Yaskawa INFORM job: u_profile_cylinder_program.JBI

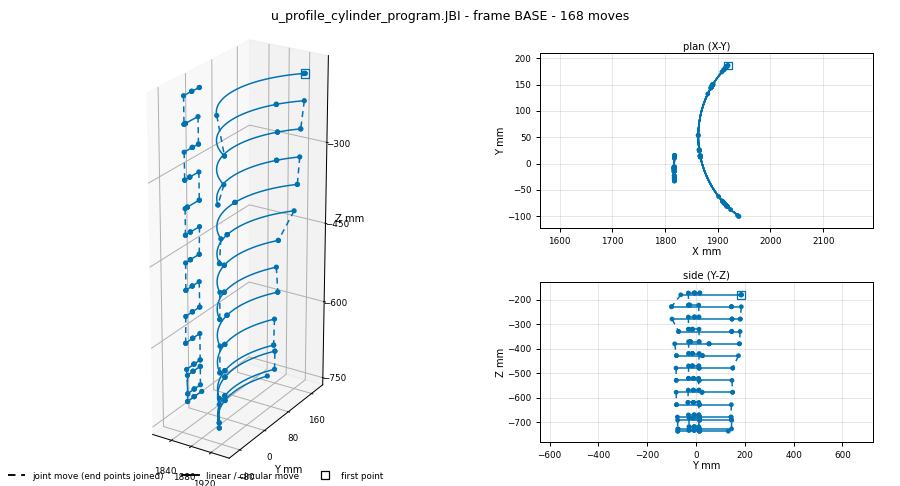
[picture p0: tool path of u_profile_cylinder_program.JBI in frame BASE, 168 of 229 moves have a stored position in this frame; points joined in program order, loops and branches not executed]
/JOB
//NAME u_profile_cylinder_program
//POS
///NPOS 224,0,224,0,0,0
///TOOL 0
///POSTYPE BASE
///RECTAN
///RCONF 0,0,0,0,0,0,0,0,0,0,0,0,0,0,0,0,0,0,0,0,0,0,0,0
C00000=1919.318375,186.161452,-178.861000,134.506550,-89.999999,5.000000
C00001=1919.318375,186.161452,-178.861000,134.506550,-89.999999,5.000000
C00002=1918.589363,185.440980,-178.861000,134.818396,-90.000000,5.000000
C00003=1917.365275,184.213378,-178.861000,135.345852,-89.999999,5.000000
C00004=1917.365275,184.213378,-178.861000,135.345852,-89.999999,5.000000
C00005=1917.365275,184.213378,-178.861000,135.345852,-89.999999,5.000000
C00006=1888.696320,146.804587,-178.861000,149.723241,-90.000000,5.000000
C00007=1901.530648,-62.264651,-178.861000,-142.697519,-90.000000,5.000000
C00008=1940.003397,-100.029578,-227.659000,-126.238595,-90.000000,5.000000
C00009=1940.003397,-100.029578,-227.659000,-126.238595,-90.000000,5.000000
C00010=1900.428189,-60.802911,-227.659000,-143.254569,-90.000000,5.000000
C00011=1887.843950,145.329282,-227.659000,150.241639,-90.000000,5.000000
C00012=1887.843950,145.329282,-227.659000,150.241639,-90.000000,5.000000
C00013=1887.843950,145.329282,-227.659000,150.241639,-90.000000,5.000000
C00014=1916.985731,183.828118,-227.659000,135.510396,-90.000000,5.000000
C00015=1918.736080,185.586610,-227.659000,134.755500,-90.000000,5.000000
C00016=1914.779750,181.544281,-278.103500,136.476486,-90.000000,5.000000
C00017=1914.779750,181.544281,-278.103500,136.476486,-90.000000,5.000000
C00018=1892.910079,153.679854,-278.103500,147.269621,-90.000000,5.000000
C00019=1889.143474,147.566403,-278.103500,149.454479,-90.000000,5.000000
C00020=1889.143474,147.566403,-278.103500,149.454479,-90.000000,5.000000
C00021=1889.143474,147.566403,-278.103500,149.454479,-90.000000,5.000000
C00022=1888.389247,146.276640,-278.103500,149.909065,-89.999999,5.000000
C00023=1937.546390,-98.197860,-278.103500,-127.171032,-89.999999,5.000000
C00024=1908.746745,-71.161367,-329.209500,-139.211685,-90.000000,5.000000
C00025=1908.746745,-71.161367,-329.209500,-139.211685,-90.000000,5.000000
C00026=1863.944997,70.602477,-329.209500,174.287971,-90.000000,5.000000
C00027=1888.494246,146.457607,-329.209500,149.845409,-90.000000,5.000000
C00028=1888.494246,146.457607,-329.209500,149.845409,-90.000000,5.000000
C00029=1888.494246,146.457607,-329.209500,149.845409,-90.000000,5.000000
C00030=1912.550325,179.155729,-329.209500,137.470595,-90.000000,5.000000
C00031=1913.986749,180.704173,-329.209500,136.827978,-90.000000,5.000000
C00032=1911.467631,177.965220,-379.550000,137.960200,-89.999999,5.000000
C00033=1911.467631,177.965220,-379.550000,137.960200,-89.999999,5.000000
C00034=1880.825526,131.812975,-379.550000,154.876624,-90.000000,5.000000
C00035=1863.018641,53.669024,-379.550000,175.000000,-90.000000,5.000000
C00036=1863.018641,53.669024,-379.550000,175.000000,-90.000000,5.000000
C00037=1863.018641,53.669024,-379.550000,175.000000,-90.000000,5.000000
C00038=1873.111078,-8.987699,-379.550000,-161.148807,-90.000000,5.000000
C00039=1924.416941,-87.270246,-379.550000,-132.370057,-90.000000,5.000000
C00040=1916.910765,-80.032620,-428.210500,-135.542952,-89.999999,5.000000
C00041=1916.910765,-80.032620,-428.210500,-135.542952,-89.999999,5.000000
C00042=1880.533893,-27.468951,-428.210500,-155.086432,-90.000000,5.000000
C00043=1864.757197,26.266217,-428.210500,-172.188992,-90.000000,5.000000
C00044=1864.757197,26.266217,-428.210500,-172.188992,-90.000000,5.000000
C00045=1864.757197,26.266217,-428.210500,-172.188992,-90.000000,5.000000
C00046=1866.619713,88.554638,-428.210500,168.763556,-90.000000,5.000000
C00047=1907.955855,173.957872,-428.210500,139.581419,-90.000000,5.000000
C00048=1890.844588,150.392245,-479.170000,148.450933,-90.000000,5.000000
C00049=1890.844588,150.392245,-479.170000,148.450933,-90.000000,5.000000
C00050=1866.110873,85.893326,-479.170000,169.587940,-90.000000,5.000000
C00051=1867.114547,12.756098,-479.170000,-168.015481,-90.000000,5.000000
C00052=1867.114547,12.756098,-479.170000,-168.015481,-90.000000,5.000000
C00053=1867.114547,12.756098,-479.170000,-168.015481,-90.000000,5.000000
C00054=1885.121266,-36.678278,-479.170000,-151.955707,-89.999999,5.000000
C00055=1918.627673,-81.759895,-479.170000,-134.801966,-90.000000,5.000000
C00056=1917.564533,-80.695611,-529.349500,-135.259659,-90.000000,5.000000
C00057=1917.564533,-80.695611,-529.349500,-135.259659,-90.000000,5.000000
C00058=1884.758137,-35.993208,-529.349500,-152.191612,-89.999999,5.000000
C00059=1867.109072,12.781899,-529.349500,-168.023506,-89.999999,5.000000
C00060=1867.109072,12.781899,-529.349500,-168.023506,-89.999999,5.000000
C00061=1867.109072,12.781899,-529.349500,-168.023506,-89.999999,5.000000
C00062=1865.977888,85.161474,-529.349500,169.814254,-90.000000,5.000000
C00063=1889.033377,147.379588,-529.349500,149.520454,-90.000000,5.000000
C00064=1890.657657,150.087139,-578.090000,148.559800,-89.999999,5.000000
C00065=1890.657657,150.087139,-578.090000,148.559800,-89.999999,5.000000
C00066=1866.130659,86.000828,-578.090000,169.554683,-90.000000,5.000000
C00067=1865.001154,24.546756,-578.090000,-171.660601,-90.000000,5.000000
C00068=1865.001154,24.546756,-578.090000,-171.660601,-90.000000,5.000000
C00069=1865.001154,24.546756,-578.090000,-171.660601,-90.000000,5.000000
C00070=1880.545792,-27.494565,-578.090000,-155.077839,-89.999999,5.000000
C00071=1918.072525,-81.206271,-578.090000,-135.040507,-90.000000,5.000000
C00072=1916.577251,-79.691863,-629.004000,-135.688022,-90.000000,5.000000
C00073=1916.577251,-79.691863,-629.004000,-135.688022,-90.000000,5.000000
C00074=1884.660871,-35.808545,-629.004000,-152.255114,-90.000000,5.000000
C00075=1866.788899,14.322936,-629.004000,-168.502384,-90.000000,5.000000
C00076=1866.788899,14.322936,-629.004000,-168.502384,-90.000000,5.000000
C00077=1866.788899,14.322936,-629.004000,-168.502384,-90.000000,5.000000
C00078=1866.111622,85.897399,-629.004000,169.586680,-90.000000,5.000000
C00079=1887.536562,144.789584,-629.004000,150.430609,-90.000000,5.000000
C00080=1886.887686,143.636513,-679.693000,150.833168,-89.999999,5.000000
C00081=1886.887686,143.636513,-679.693000,150.833168,-89.999999,5.000000
C00082=1865.941224,84.956765,-679.693000,169.877528,-89.999999,5.000000
C00083=1866.729376,14.616759,-679.693000,-168.593596,-90.000000,5.000000
C00084=1866.729376,14.616759,-679.693000,-168.593596,-90.000000,5.000000
C00085=1866.729376,14.616759,-679.693000,-168.593596,-90.000000,5.000000
C00086=1884.804416,-36.080897,-679.693000,-152.161445,-89.999999,5.000000
C00087=1913.224618,-76.167805,-679.693000,-137.167966,-90.000000,5.000000
C00088=1911.184789,-73.931681,-728.214500,-138.088869,-90.000000,5.000000
C00089=1911.184789,-73.931681,-728.214500,-138.088869,-90.000000,5.000000
C00090=1884.746150,-35.970477,-728.214500,-152.199431,-89.999999,5.000000
C00091=1866.919433,13.686824,-728.214500,-168.304812,-90.000000,5.000000
C00092=1866.919433,13.686824,-728.214500,-168.304812,-90.000000,5.000000
C00093=1866.919433,13.686824,-728.214500,-168.304812,-90.000000,5.000000
C00094=1865.765968,83.959631,-728.214500,170.185559,-89.999999,5.000000
C00095=1887.960264,145.532429,-728.214500,150.170417,-90.000000,5.000000
C00096=1888.186604,145.926067,-692.282460,175.000000,-60.000000,-29.967735
C00097=1888.186604,145.926067,-692.282460,175.000000,-60.000000,-29.967735
C00098=1865.952407,85.019339,-692.282460,175.000000,-60.000000,-10.141812
C00099=1866.711119,14.707370,-692.282460,175.000000,-60.000000,11.378282
C00100=1866.711119,14.707370,-692.282460,175.000000,-60.000000,11.378282
C00101=1866.711119,14.707370,-692.282460,175.000000,-60.000000,11.378282
C00102=1884.830220,-36.129742,-692.282460,-175.000000,-60.000000,27.855362
C00103=1912.302833,-75.166247,-692.282460,-175.000000,-60.000000,42.417891
C00104=1911.869257,-74.690086,-737.636460,175.000000,-60.000000,42.221957
C00105=1911.869257,-74.690086,-737.636460,175.000000,-60.000000,42.221957
C00106=1884.879767,-36.223432,-737.636460,175.000000,-60.000000,27.887609
C00107=1866.818502,14.177698,-737.636460,175.000000,-60.000000,11.542714
C00108=1866.818502,14.177698,-737.636460,175.000000,-60.000000,11.542714
C00109=1866.818502,14.177698,-737.636460,175.000000,-60.000000,11.542714
C00110=1864.683098,76.906826,-737.636460,175.000000,-60.000000,-7.643334
C00111=1881.053412,132.297152,-737.636460,175.000000,-60.000000,-25.286189
C00112=1817.990504,15.588637,-171.217500,175.000000,-89.999999,5.000000
C00113=1817.990504,15.588637,-171.217500,175.000000,-89.999999,5.000000
C00114=1817.535552,3.881759,-171.217500,175.000000,-90.000000,5.000000
C00115=1817.349789,-6.442676,-171.217500,175.000000,-90.000000,5.000000
C00116=1817.349789,-6.442676,-171.217500,175.000000,-90.000000,5.000000
C00117=1817.349789,-6.442676,-171.217500,175.000000,-90.000000,5.000000
C00118=1817.526814,-25.140198,-171.217500,-175.000000,-90.000000,5.000000
C00119=1817.723727,-31.135669,-171.217500,-175.000000,-90.000000,5.000000
C00120=1817.711525,-30.816430,-220.926500,-175.000000,-90.000000,5.000000
C00121=1817.711525,-30.816430,-220.926500,-175.000000,-90.000000,5.000000
C00122=1817.677190,-29.889507,-220.926500,-175.000000,-89.999999,5.000000
C00123=1817.559266,-26.288875,-220.926500,-175.000000,-89.999999,5.000000
C00124=1817.559266,-26.288875,-220.926500,-175.000000,-89.999999,5.000000
C00125=1817.559266,-26.288875,-220.926500,-175.000000,-89.999999,5.000000
C00126=1817.458554,-22.357350,-220.926500,-175.000000,-90.000000,5.000000
C00127=1817.791962,11.259122,-220.926500,175.000000,-89.999999,5.000000
C00128=1817.818806,11.892960,-269.769000,175.000000,-90.000000,5.000000
C00129=1817.818806,11.892960,-269.769000,175.000000,-90.000000,5.000000
C00130=1817.515491,3.140532,-269.769000,175.000000,-90.000000,5.000000
C00131=1817.353005,-6.067748,-269.769000,175.000000,-89.999999,5.000000
C00132=1817.353005,-6.067748,-269.769000,175.000000,-89.999999,5.000000
C00133=1817.353005,-6.067748,-269.769000,175.000000,-89.999999,5.000000
C00134=1817.536459,-25.490982,-269.769000,-175.000000,-89.999999,5.000000
C00135=1817.725812,-31.189730,-269.769000,-175.000000,-89.999999,5.000000
C00136=1817.698334,-30.465502,-319.757000,-175.000000,-89.999999,5.000000
C00137=1817.698334,-30.465502,-319.757000,-175.000000,-89.999999,5.000000
C00138=1817.564494,-26.466058,-319.757000,-175.000000,-89.999999,5.000000
C00139=1817.346049,-14.652350,-319.757000,-175.000000,-90.000000,5.000000
C00140=1817.346049,-14.652350,-319.757000,-175.000000,-90.000000,5.000000
C00141=1817.346049,-14.652350,-319.757000,-175.000000,-90.000000,5.000000
C00142=1817.456468,0.685090,-319.757000,175.000000,-90.000000,5.000000
C00143=1817.843348,12.457295,-319.757000,175.000000,-89.999999,5.000000
C00144=1817.862419,12.886540,-370.985000,175.000000,-89.999999,5.000000
C00145=1817.862419,12.886540,-370.985000,175.000000,-89.999999,5.000000
C00146=1817.718241,9.416200,-370.985000,175.000000,-89.999999,5.000000
C00147=1817.468232,-22.791229,-370.985000,-175.000000,-90.000000,5.000000
C00148=1817.468232,-22.791229,-370.985000,-175.000000,-90.000000,5.000000
C00149=1817.468232,-22.791229,-370.985000,-175.000000,-90.000000,5.000000
C00150=1817.608303,-27.878641,-370.985000,-175.000000,-90.000000,5.000000
C00151=1817.689997,-30.240415,-370.985000,-175.000000,-90.000000,5.000000
C00152=1817.677729,-29.904397,-419.370500,-175.000000,-90.000000,5.000000
C00153=1817.677729,-29.904397,-419.370500,-175.000000,-90.000000,5.000000
C00154=1817.565488,-26.499532,-419.370500,-175.000000,-90.000000,5.000000
C00155=1817.344102,-14.376187,-419.370500,-175.000000,-89.999999,5.000000
C00156=1817.344102,-14.376187,-419.370500,-175.000000,-89.999999,5.000000
C00157=1817.344102,-14.376187,-419.370500,-175.000000,-89.999999,5.000000
C00158=1817.497248,2.430436,-419.370500,175.000000,-89.999999,5.000000
C00159=1817.865089,12.946001,-419.370500,175.000000,-90.000000,5.000000
C00160=1817.804165,11.549491,-470.057500,175.000000,-90.000000,5.000000
C00161=1817.804165,11.549491,-470.057500,175.000000,-90.000000,5.000000
C00162=1817.398164,-2.420661,-470.057500,175.000000,-89.999999,5.000000
C00163=1817.348154,-14.930333,-470.057500,-175.000000,-89.999999,5.000000
C00164=1817.348154,-14.930333,-470.057500,-175.000000,-89.999999,5.000000
C00165=1817.348154,-14.930333,-470.057500,-175.000000,-89.999999,5.000000
C00166=1817.479346,-23.270935,-470.057500,-175.000000,-89.999999,5.000000
C00167=1817.696262,-30.409800,-470.057500,-175.000000,-90.000000,5.000000
C00168=1817.702789,-30.584713,-520.961000,-175.000000,-89.999999,5.000000
C00169=1817.702789,-30.584713,-520.961000,-175.000000,-89.999999,5.000000
C00170=1817.473301,-23.012345,-520.961000,-175.000000,-89.999999,5.000000
C00171=1817.332146,-10.303971,-520.961000,175.000000,-89.999999,5.000000
C00172=1817.332146,-10.303971,-520.961000,175.000000,-89.999999,5.000000
C00173=1817.332146,-10.303971,-520.961000,175.000000,-89.999999,5.000000
C00174=1817.481924,1.803009,-520.961000,175.000000,-90.000000,5.000000
C00175=1817.771654,10.767186,-520.961000,175.000000,-90.000000,5.000000
C00176=1817.807943,11.638625,-569.380500,175.000000,-89.999999,5.000000
C00177=1817.807943,11.638625,-569.380500,175.000000,-89.999999,5.000000
C00178=1817.492353,2.233288,-569.380500,175.000000,-90.000000,5.000000
C00179=1817.332011,-10.484289,-569.380500,175.000000,-89.999999,5.000000
C00180=1817.332011,-10.484289,-569.380500,175.000000,-89.999999,5.000000
C00181=1817.332011,-10.484289,-569.380500,175.000000,-89.999999,5.000000
C00182=1817.402898,-19.449712,-569.380500,-175.000000,-90.000000,5.000000
C00183=1817.753185,-31.886429,-569.380500,-175.000000,-90.000000,5.000000
C00184=1817.797491,-32.967741,-619.760000,-175.000000,-90.000000,5.000000
C00185=1817.797491,-32.967741,-619.760000,-175.000000,-90.000000,5.000000
C00186=1817.408869,-19.806675,-619.760000,-175.000000,-90.000000,5.000000
C00187=1817.332035,-10.445182,-619.760000,175.000000,-90.000000,5.000000
C00188=1817.332035,-10.445182,-619.760000,175.000000,-90.000000,5.000000
C00189=1817.332035,-10.445182,-619.760000,175.000000,-90.000000,5.000000
C00190=1817.487025,2.015284,-619.760000,175.000000,-90.000000,5.000000
C00191=1817.799497,11.438868,-619.760000,175.000000,-90.000000,5.000000
C00192=1817.816514,11.839522,-670.886500,175.000000,-90.000000,5.000000
C00193=1817.816514,11.839522,-670.886500,175.000000,-90.000000,5.000000
C00194=1817.497087,2.424002,-670.886500,175.000000,-89.999999,5.000000
C00195=1817.343542,-7.283868,-670.886500,175.000000,-90.000000,5.000000
C00196=1817.343542,-7.283868,-670.886500,175.000000,-90.000000,5.000000
C00197=1817.343542,-7.283868,-670.886500,175.000000,-90.000000,5.000000
C00198=1817.403330,-19.476025,-670.886500,-175.000000,-89.999999,5.000000
C00199=1817.714379,-30.891550,-670.886500,-175.000000,-90.000000,5.000000
C00200=1817.617890,-28.172449,-719.382000,-175.000000,-89.999999,5.000000
C00201=1817.617890,-28.172449,-719.382000,-175.000000,-89.999999,5.000000
C00202=1817.404390,-19.540283,-719.382000,-175.000000,-90.000000,5.000000
C00203=1817.344900,-7.084679,-719.382000,175.000000,-89.999999,5.000000
C00204=1817.344900,-7.084679,-719.382000,175.000000,-89.999999,5.000000
C00205=1817.344900,-7.084679,-719.382000,175.000000,-89.999999,5.000000
C00206=1817.490538,2.159410,-719.382000,175.000000,-89.999999,5.000000
C00207=1817.819284,11.904095,-719.382000,175.000000,-89.999999,5.000000
C00208=1817.821861,11.963975,-683.466460,175.000000,-60.000000,-5.000000
C00209=1817.821861,11.963975,-683.466460,175.000000,-60.000000,-5.000000
C00210=1817.474996,1.508823,-683.466460,-175.000000,-60.000000,-5.000000
C00211=1817.332124,-10.329006,-683.466460,175.000000,-60.000000,-5.000000
C00212=1817.332124,-10.329006,-683.466460,175.000000,-60.000000,-5.000000
C00213=1817.332124,-10.329006,-683.466460,175.000000,-60.000000,-5.000000
C00214=1817.403522,-19.487738,-683.466460,175.000000,-60.000000,5.000000
C00215=1817.622059,-28.298669,-683.466460,175.000000,-60.000000,5.000000
C00216=1817.637760,-28.766095,-734.096960,175.000000,-60.000000,5.000000
C00217=1817.637760,-28.766095,-734.096960,175.000000,-60.000000,5.000000
C00218=1817.405775,-19.623546,-734.096960,-175.000000,-60.000000,5.000000
C00219=1817.341568,-7.595472,-734.096960,-175.000000,-60.000000,-5.000000
C00220=1817.341568,-7.595472,-734.096960,-175.000000,-60.000000,-5.000000
C00221=1817.341568,-7.595472,-734.096960,-175.000000,-60.000000,-5.000000
C00222=1817.484869,1.925964,-734.096960,-175.000000,-60.000000,-5.000000
C00223=1817.997034,15.719000,-734.096960,175.000000,-60.000000,-5.000000
///POSTYPE PULSE
///PULSE
EX00000=261120.0
EX00001=362496.0
///POSTYPE PULSE
///PULSE
EC00000=261120.0
EC00001=261120.0
EC00002=261120.0
EC00003=261120.0
EC00004=261120.0
EC00005=261120.0
EC00006=261120.0
EC00007=261120.0
EC00008=261120.0
EC00009=261120.0
EC00010=261120.0
EC00011=261120.0
EC00012=261120.0
EC00013=261120.0
EC00014=261120.0
EC00015=261120.0
EC00016=261120.0
EC00017=261120.0
EC00018=261120.0
EC00019=261120.0
EC00020=261120.0
EC00021=261120.0
EC00022=261120.0
EC00023=261120.0
EC00024=261120.0
EC00025=261120.0
EC00026=261120.0
EC00027=261120.0
EC00028=261120.0
EC00029=261120.0
EC00030=261120.0
EC00031=261120.0
EC00032=261120.0
EC00033=261120.0
EC00034=261120.0
EC00035=261120.0
EC00036=261120.0
EC00037=261120.0
EC00038=261120.0
EC00039=261120.0
EC00040=261120.0
EC00041=261120.0
EC00042=261120.0
EC00043=261120.0
EC00044=261120.0
EC00045=261120.0
EC00046=261120.0
EC00047=261120.0
EC00048=261120.0
EC00049=261120.0
EC00050=261120.0
EC00051=261120.0
EC00052=261120.0
EC00053=261120.0
EC00054=261120.0
EC00055=261120.0
EC00056=261120.0
EC00057=261120.0
EC00058=261120.0
EC00059=261120.0
EC00060=261120.0
EC00061=261120.0
EC00062=261120.0
EC00063=261120.0
EC00064=261120.0
EC00065=261120.0
EC00066=261120.0
EC00067=261120.0
EC00068=261120.0
EC00069=261120.0
EC00070=261120.0
EC00071=261120.0
EC00072=261120.0
EC00073=261120.0
EC00074=261120.0
EC00075=261120.0
EC00076=261120.0
EC00077=261120.0
EC00078=261120.0
EC00079=261120.0
EC00080=261120.0
EC00081=261120.0
EC00082=261120.0
EC00083=261120.0
EC00084=261120.0
EC00085=261120.0
EC00086=261120.0
EC00087=261120.0
EC00088=261120.0
EC00089=261120.0
EC00090=261120.0
EC00091=261120.0
EC00092=261120.0
EC00093=261120.0
EC00094=261120.0
EC00095=261120.0
EC00096=261120.0
EC00097=261120.0
EC00098=261120.0
EC00099=261120.0
EC00100=261120.0
EC00101=261120.0
EC00102=261120.0
EC00103=261120.0
EC00104=261120.0
EC00105=261120.0
EC00106=261120.0
EC00107=261120.0
EC00108=261120.0
EC00109=261120.0
EC00110=261120.0
EC00111=261120.0
EC00112=362496.0
EC00113=362496.0
EC00114=362496.0
EC00115=362496.0
EC00116=362496.0
EC00117=362496.0
EC00118=362496.0
EC00119=362496.0
EC00120=362496.0
EC00121=362496.0
EC00122=362496.0
EC00123=362496.0
EC00124=362496.0
EC00125=362496.0
EC00126=362496.0
EC00127=362496.0
EC00128=362496.0
EC00129=362496.0
EC00130=362496.0
EC00131=362496.0
EC00132=362496.0
EC00133=362496.0
EC00134=362496.0
EC00135=362496.0
EC00136=362496.0
EC00137=362496.0
EC00138=362496.0
EC00139=362496.0
EC00140=362496.0
EC00141=362496.0
EC00142=362496.0
EC00143=362496.0
EC00144=362496.0
EC00145=362496.0
EC00146=362496.0
EC00147=362496.0
EC00148=362496.0
EC00149=362496.0
EC00150=362496.0
EC00151=362496.0
EC00152=362496.0
EC00153=362496.0
EC00154=362496.0
EC00155=362496.0
EC00156=362496.0
EC00157=362496.0
EC00158=362496.0
EC00159=362496.0
EC00160=362496.0
EC00161=362496.0
EC00162=362496.0
EC00163=362496.0
EC00164=362496.0
EC00165=362496.0
EC00166=362496.0
EC00167=362496.0
EC00168=362496.0
EC00169=362496.0
EC00170=362496.0
EC00171=362496.0
EC00172=362496.0
EC00173=362496.0
EC00174=362496.0
EC00175=362496.0
EC00176=362496.0
EC00177=362496.0
EC00178=362496.0
EC00179=362496.0
EC00180=362496.0
EC00181=362496.0
EC00182=362496.0
EC00183=362496.0
EC00184=362496.0
EC00185=362496.0
EC00186=362496.0
EC00187=362496.0
EC00188=362496.0
EC00189=362496.0
EC00190=362496.0
EC00191=362496.0
EC00192=362496.0
EC00193=362496.0
EC00194=362496.0
EC00195=362496.0
EC00196=362496.0
EC00197=362496.0
EC00198=362496.0
EC00199=362496.0
EC00200=362496.0
EC00201=362496.0
EC00202=362496.0
EC00203=362496.0
EC00204=362496.0
EC00205=362496.0
EC00206=362496.0
EC00207=362496.0
EC00208=362496.0
EC00209=362496.0
EC00210=362496.0
EC00211=362496.0
EC00212=362496.0
EC00213=362496.0
EC00214=362496.0
EC00215=362496.0
EC00216=362496.0
EC00217=362496.0
EC00218=362496.0
EC00219=362496.0
EC00220=362496.0
EC00221=362496.0
EC00222=362496.0
EC00223=362496.0
//INST
///DATE 2023/08/16 15:26
///ATTR SC,RW,RJ
////FRAME BASE
///GROUP1 RB1,ST1
NOP
MOVJ P009 EX000 VJ=15.00
MOVJ C00000 EC00000 VJ=15.0
CALL JOB:SPYON
MOVC C00001 EC00001 V=150.0
MOVC C00002 EC00002 V=150.0
MOVC C00003 EC00003 V=150.0
MOVJ C00004 EC00004 VJ=15.0
MOVC C00005 EC00005 V=150.0
MOVC C00006 EC00006 V=150.0
MOVC C00007 EC00007 V=150.0
MOVJ C00008 EC00008 VJ=15.0
MOVC C00009 EC00009 V=150.0
MOVC C00010 EC00010 V=150.0
MOVC C00011 EC00011 V=150.0
MOVJ C00012 EC00012 VJ=15.0
MOVC C00013 EC00013 V=150.0
MOVC C00014 EC00014 V=150.0
MOVC C00015 EC00015 V=150.0
MOVJ C00016 EC00016 VJ=15.0
MOVC C00017 EC00017 V=150.0
MOVC C00018 EC00018 V=150.0
MOVC C00019 EC00019 V=150.0
MOVJ C00020 EC00020 VJ=15.0
MOVC C00021 EC00021 V=150.0
MOVC C00022 EC00022 V=150.0
MOVC C00023 EC00023 V=150.0
MOVJ C00024 EC00024 VJ=15.0
MOVC C00025 EC00025 V=150.0
MOVC C00026 EC00026 V=150.0
MOVC C00027 EC00027 V=150.0
MOVJ C00028 EC00028 VJ=15.0
MOVC C00029 EC00029 V=150.0
MOVC C00030 EC00030 V=150.0
MOVC C00031 EC00031 V=150.0
MOVJ C00032 EC00032 VJ=15.0
MOVC C00033 EC00033 V=150.0
MOVC C00034 EC00034 V=150.0
MOVC C00035 EC00035 V=150.0
MOVJ C00036 EC00036 VJ=15.0
MOVC C00037 EC00037 V=150.0
MOVC C00038 EC00038 V=150.0
MOVC C00039 EC00039 V=150.0
MOVJ C00040 EC00040 VJ=15.0
MOVC C00041 EC00041 V=150.0
MOVC C00042 EC00042 V=150.0
MOVC C00043 EC00043 V=150.0
MOVJ C00044 EC00044 VJ=15.0
MOVC C00045 EC00045 V=150.0
MOVC C00046 EC00046 V=150.0
MOVC C00047 EC00047 V=150.0
MOVJ C00048 EC00048 VJ=15.0
MOVC C00049 EC00049 V=150.0
MOVC C00050 EC00050 V=150.0
MOVC C00051 EC00051 V=150.0
MOVJ C00052 EC00052 VJ=15.0
MOVC C00053 EC00053 V=150.0
MOVC C00054 EC00054 V=150.0
MOVC C00055 EC00055 V=150.0
MOVJ C00056 EC00056 VJ=15.0
MOVC C00057 EC00057 V=150.0
MOVC C00058 EC00058 V=150.0
MOVC C00059 EC00059 V=150.0
MOVJ C00060 EC00060 VJ=15.0
MOVC C00061 EC00061 V=150.0
MOVC C00062 EC00062 V=150.0
MOVC C00063 EC00063 V=150.0
MOVJ C00064 EC00064 VJ=15.0
MOVC C00065 EC00065 V=150.0
MOVC C00066 EC00066 V=150.0
MOVC C00067 EC00067 V=150.0
MOVJ C00068 EC00068 VJ=15.0
MOVC C00069 EC00069 V=150.0
MOVC C00070 EC00070 V=150.0
MOVC C00071 EC00071 V=150.0
MOVJ C00072 EC00072 VJ=15.0
MOVC C00073 EC00073 V=150.0
MOVC C00074 EC00074 V=150.0
MOVC C00075 EC00075 V=150.0
MOVJ C00076 EC00076 VJ=15.0
MOVC C00077 EC00077 V=150.0
MOVC C00078 EC00078 V=150.0
MOVC C00079 EC00079 V=150.0
MOVJ C00080 EC00080 VJ=15.0
MOVC C00081 EC00081 V=150.0
MOVC C00082 EC00082 V=150.0
MOVC C00083 EC00083 V=150.0
MOVJ C00084 EC00084 VJ=15.0
MOVC C00085 EC00085 V=150.0
MOVC C00086 EC00086 V=150.0
MOVC C00087 EC00087 V=150.0
MOVJ C00088 EC00088 VJ=15.0
MOVC C00089 EC00089 V=150.0
MOVC C00090 EC00090 V=150.0
MOVC C00091 EC00091 V=150.0
MOVJ C00092 EC00092 VJ=15.0
MOVC C00093 EC00093 V=150.0
MOVC C00094 EC00094 V=150.0
MOVC C00095 EC00095 V=150.0
MOVJ C00096 EC00096 VJ=15.0
MOVC C00097 EC00097 V=150.0
MOVC C00098 EC00098 V=150.0
MOVC C00099 EC00099 V=150.0
MOVJ C00100 EC00100 VJ=15.0
MOVC C00101 EC00101 V=150.0
MOVC C00102 EC00102 V=150.0
MOVC C00103 EC00103 V=150.0
MOVJ C00104 EC00104 VJ=15.0
MOVC C00105 EC00105 V=150.0
MOVC C00106 EC00106 V=150.0
MOVC C00107 EC00107 V=150.0
MOVJ C00108 EC00108 VJ=15.0
MOVC C00109 EC00109 V=150.0
MOVC C00110 EC00110 V=150.0
MOVC C00111 EC00111 V=150.0
CALL JOB:SPYOF
MOVJ P009 VJ=15.00
MOVL P009 EX00000 V=150.0
MOVJ C00112 EC00112 VJ=15.0
CALL JOB:SPYON
MOVC C00113 EC00113 V=150.0
MOVC C00114 EC00114 V=150.0
MOVC C00115 EC00115 V=150.0
MOVJ C00116 EC00116 VJ=15.0
MOVC C00117 EC00117 V=150.0
MOVC C00118 EC00118 V=150.0
MOVC C00119 EC00119 V=150.0
MOVJ C00120 EC00120 VJ=15.0
MOVC C00121 EC00121 V=150.0
MOVC C00122 EC00122 V=150.0
MOVC C00123 EC00123 V=150.0
MOVJ C00124 EC00124 VJ=15.0
MOVC C00125 EC00125 V=150.0
MOVC C00126 EC00126 V=150.0
MOVC C00127 EC00127 V=150.0
MOVJ C00128 EC00128 VJ=15.0
MOVC C00129 EC00129 V=150.0
MOVC C00130 EC00130 V=150.0
MOVC C00131 EC00131 V=150.0
MOVJ C00132 EC00132 VJ=15.0
MOVC C00133 EC00133 V=150.0
MOVC C00134 EC00134 V=150.0
MOVC C00135 EC00135 V=150.0
MOVJ C00136 EC00136 VJ=15.0
MOVC C00137 EC00137 V=150.0
MOVC C00138 EC00138 V=150.0
MOVC C00139 EC00139 V=150.0
MOVJ C00140 EC00140 VJ=15.0
MOVC C00141 EC00141 V=150.0
MOVC C00142 EC00142 V=150.0
MOVC C00143 EC00143 V=150.0
MOVJ C00144 EC00144 VJ=15.0
MOVC C00145 EC00145 V=150.0
MOVC C00146 EC00146 V=150.0
MOVC C00147 EC00147 V=150.0
MOVJ C00148 EC00148 VJ=15.0
MOVC C00149 EC00149 V=150.0
MOVC C00150 EC00150 V=150.0
MOVC C00151 EC00151 V=150.0
MOVJ C00152 EC00152 VJ=15.0
MOVC C00153 EC00153 V=150.0
MOVC C00154 EC00154 V=150.0
MOVC C00155 EC00155 V=150.0
MOVJ C00156 EC00156 VJ=15.0
MOVC C00157 EC00157 V=150.0
MOVC C00158 EC00158 V=150.0
MOVC C00159 EC00159 V=150.0
MOVJ C00160 EC00160 VJ=15.0
MOVC C00161 EC00161 V=150.0
MOVC C00162 EC00162 V=150.0
MOVC C00163 EC00163 V=150.0
MOVJ C00164 EC00164 VJ=15.0
MOVC C00165 EC00165 V=150.0
MOVC C00166 EC00166 V=150.0
MOVC C00167 EC00167 V=150.0
MOVJ C00168 EC00168 VJ=15.0
MOVC C00169 EC00169 V=150.0
MOVC C00170 EC00170 V=150.0
MOVC C00171 EC00171 V=150.0
MOVJ C00172 EC00172 VJ=15.0
MOVC C00173 EC00173 V=150.0
MOVC C00174 EC00174 V=150.0
MOVC C00175 EC00175 V=150.0
MOVJ C00176 EC00176 VJ=15.0
MOVC C00177 EC00177 V=150.0
MOVC C00178 EC00178 V=150.0
MOVC C00179 EC00179 V=150.0
MOVJ C00180 EC00180 VJ=15.0
MOVC C00181 EC00181 V=150.0
MOVC C00182 EC00182 V=150.0
MOVC C00183 EC00183 V=150.0
MOVJ C00184 EC00184 VJ=15.0
MOVC C00185 EC00185 V=150.0
MOVC C00186 EC00186 V=150.0
MOVC C00187 EC00187 V=150.0
MOVJ C00188 EC00188 VJ=15.0
MOVC C00189 EC00189 V=150.0
MOVC C00190 EC00190 V=150.0
MOVC C00191 EC00191 V=150.0
MOVJ C00192 EC00192 VJ=15.0
MOVC C00193 EC00193 V=150.0
MOVC C00194 EC00194 V=150.0
MOVC C00195 EC00195 V=150.0
MOVJ C00196 EC00196 VJ=15.0
MOVC C00197 EC00197 V=150.0
MOVC C00198 EC00198 V=150.0
MOVC C00199 EC00199 V=150.0
MOVJ C00200 EC00200 VJ=15.0
MOVC C00201 EC00201 V=150.0
MOVC C00202 EC00202 V=150.0
MOVC C00203 EC00203 V=150.0
MOVJ C00204 EC00204 VJ=15.0
MOVC C00205 EC00205 V=150.0
MOVC C00206 EC00206 V=150.0
MOVC C00207 EC00207 V=150.0
MOVJ C00208 EC00208 VJ=15.0
MOVC C00209 EC00209 V=150.0
MOVC C00210 EC00210 V=150.0
MOVC C00211 EC00211 V=150.0
MOVJ C00212 EC00212 VJ=15.0
MOVC C00213 EC00213 V=150.0
MOVC C00214 EC00214 V=150.0
MOVC C00215 EC00215 V=150.0
MOVJ C00216 EC00216 VJ=15.0
MOVC C00217 EC00217 V=150.0
MOVC C00218 EC00218 V=150.0
MOVC C00219 EC00219 V=150.0
MOVJ C00220 EC00220 VJ=15.0
MOVC C00221 EC00221 V=150.0
MOVC C00222 EC00222 V=150.0
MOVC C00223 EC00223 V=150.0
CALL JOB:SPYOF
MOVJ P009 VJ=15.00
MOVL P009 EX00001 V=150.0
END
